(* IEC 61131-3 sources: Lasal/CPU_5344_V01/Class/loaderUnitSettingsMpsControl, 1 file *)

(* ---- loaderUnitSettingsMpsControl.st ---- *)
(*!
<Class
	Name               = "loaderUnitSettingsMpsControl"
	Revision           = "1.0"
	RealtimeTask       = "false"
	CyclicTask         = "false"
	BackgroundTask     = "false"
	Sigmatek           = "false"
	OSInterface        = "false"
	HighPriority       = "false"
	Automatic          = "false"
	UpdateMode         = "Prescan"
	SharedCommandTable = "true"
	Objectsize         = "(284,120)">
	<Channels>
		<Server Name="setting1" Visualized="true" Initialize="false" WriteProtected="false" Retentive="false" Comment="position in x-direction (1/10mm)"/>
		<Server Name="setting2" Visualized="true" Initialize="true" DefValue="1" WriteProtected="false" Retentive="false" Comment="&apos;is load-in&apos; (value  1, load in unit; value 0, push out unit)"/>
		<Server Name="setting3" Visualized="true" Initialize="true" WriteProtected="false" Retentive="false" Comment="&apos;can do waste&apos; (0 not possible, 1 possible)"/>
		<Server Name="setting4" Visualized="true" Initialize="false" WriteProtected="false" Retentive="false" Comment="amount of positions for visualization"/>
		<Client Name="iAmountOfPositions" Required="false" Internal="false"/>
		<Client Name="iOffset" Required="true" Internal="false"/>
	</Channels>
	<Network Name="loaderUnitSettingsMpsControl">
		<!-- List of Components in this network -->
		<Components>
			<Object
				Name       = "_base"
				Class      = "baseToolSettingsMpsControl"
				Position   = "(218,120)"
				Visualized = "true">
				<Channels>
					<Server Name="amountOfSettings" Value="4"/>
					<Server Name="ClassSvr"/>
					<Server Name="Name"/>
					<Server Name="plane"/>
					<Server Name="toolType" Value="1"/>
				</Channels>
			</Object>
		</Components>
		<Comments>
		</Comments>
		<!-- List of Connections in this network -->
		<Connections>
			<Connection Source="this.ClassSvr" Destination="_base.ClassSvr" Vertices="(690,210),(518,210),"/>
			<Connection Source="this.toolType" Destination="_base.toolType" Vertices="(690,270),(518,270),"/>
			<Connection Source="this.amountOfSettings" Destination="_base.amountOfSettings" Vertices="(690,450),(518,450),"/>
			<Connection Source="this.plane" Destination="_base.plane" Vertices="(690,390),(518,390),"/>
			<Connection Source="this.Name" Destination="_base.Name" Vertices="(690,330),(518,330),"/>
		</Connections>
		<!-- Headerfiles -->
		<Options>
		</Options>
	</Network>
</Class>
*)
#pragma using baseToolSettingsMpsControl

loaderUnitSettingsMpsControl : CLASS
: baseToolSettingsMpsControl
  //Servers:
	setting1 	: SvrCh_DINT;
	setting2 	: SvrCh_DINT;
	setting3 	: SvrCh_DINT;
	setting4 	: SvrCh_DINT;
  //Clients:
	iOffset 	: CltCh_DINT;
	iAmountOfPositions 	: CltCh_DINT;
  //Variables:
  //Functions:

	FUNCTION VIRTUAL GLOBAL setting1::Read
		VAR_OUTPUT
			output (EAX) 	: DINT;
		END_VAR;

	FUNCTION VIRTUAL GLOBAL setting4::Read
		VAR_OUTPUT
			output (EAX) 	: DINT;
		END_VAR;
  //Tables:
	FUNCTION @STD
		VAR_OUTPUT
			ret_code	: CONFSTATES;
		END_VAR;
	FUNCTION GLOBAL TAB @CT_;
END_CLASS;

// JdK 4-2-2020: punchToolSettingsMpsControlOld created for first test to read in settings to pc
// at this moment the class is only for storage off fixed machine data for punch tools

FUNCTION VIRTUAL GLOBAL loaderUnitSettingsMpsControl::setting1::Read
	VAR_OUTPUT
		output (EAX) 	: DINT;
	END_VAR

  iOffset:= iOffset.Read();
  setting1:= iOffset;
	output := setting1;

END_FUNCTION

FUNCTION VIRTUAL GLOBAL loaderUnitSettingsMpsControl::setting4::Read
	VAR_OUTPUT
		output (EAX) 	: DINT;
	END_VAR

  iAmountOfPositions:= iAmountOfPositions.Read();
  setting4:= iAmountOfPositions;
	output := setting4;

END_FUNCTION
